FUNCTION_BLOCK FB_OmronLD90 EXTENDS FB_ROB_AMR IMPLEMENTS 
VAR_INPUT
END_VAR
VAR_OUTPUT
END_VAR
VAR
	//Reference to Skills

END_VAR

StateMachine(); // Method in FB_Base
ComMachine();	//Method in FB_ROB
DBClient();	//Datenbank Client in FB_ROB


PiNPl(Rob:=ADR(THIS^));

METHOD ComMachine : BOOL
VAR_INPUT
END_VAR
CASE eConnectionState OF


    // =========================================================
    // DISCONNECTED
    // =========================================================

    eCommunicationState.DISCONNECTED:

       _connected := FALSE;


        // Make sure socket handle is cleared
//         hSocket


        // -----------------------------------------------------
        // Connect requested
        // -----------------------------------------------------

        IF xConnectRequest THEN

            xConnectRequest := FALSE;

            // Clear previous errors
            Error := FALSE;
            ErrorId := 0;
            SocketErrorId := 0;

            // Start FB_SocketConnect
            xSocketConnectExecute := TRUE;

            eConnectionState :=
                eCommunicationState.CONNECTING;

        END_IF;


    // =========================================================
    // CONNECTING
    // =========================================================

    eCommunicationState.CONNECTING:

        _connected := FALSE;
        


        // -----------------------------------------------------
        // Execute FB_SocketConnect
        // -----------------------------------------------------

        fbSocketConnect(
            sSrvNetId := '',
            sRemoteHost := ComConfig.sIpAddress,
            nRemotePort := ComConfig.nPort,
            bExecute := xSocketConnectExecute,
            tTimeout := ComConfig.tTimeout
        );


        // Execute must only be TRUE for one cycle
        xSocketConnectExecute := FALSE;


        // -----------------------------------------------------
        // Connection successful
        // -----------------------------------------------------

        IF NOT fbSocketConnect.bBusy
            AND NOT fbSocketConnect.bError
//             AND (fbSocketConnect.hSocket <> 0)
        THEN

            hSocket :=
                fbSocketConnect.hSocket;

            _connected := TRUE;
    

            Error := FALSE;
            ErrorId := 0;
            SocketErrorId := 0;

            eConnectionState :=
                eCommunicationState.CONNECTED;

        END_IF;


        // -----------------------------------------------------
        // Connection failed
        // -----------------------------------------------------

        IF NOT fbSocketConnect.bBusy
            AND fbSocketConnect.bError
        THEN

            _connected := FALSE;

            Error := TRUE;

            SocketErrorId :=
                fbSocketConnect.nErrId;

            ErrorId :=
                fbSocketConnect.nErrId;

//             hSocket := 0;

            eConnectionState :=
                eCommunicationState.ERROR;

        END_IF;


    // =========================================================
    // CONNECTED
    // =========================================================

    eCommunicationState.CONNECTED:

        _connected := TRUE;



        // -----------------------------------------------------
        // Disconnect requested
        // -----------------------------------------------------

        IF xDisconnectRequest THEN

            xDisconnectRequest := FALSE;


            // Start socket close
            xSocketCloseExecute := TRUE;

            eConnectionState :=
                eCommunicationState.DISCONNECTING;

        END_IF;


    // =========================================================
    // DISCONNECTING
    // =========================================================

    eCommunicationState.DISCONNECTING:

        _connected := FALSE;


        // -----------------------------------------------------
        // Execute FB_SocketClose
        // -----------------------------------------------------

        fbSocketClose(
            sSrvNetId := '',
            hSocket := hSocket,
            bExecute := xSocketCloseExecute,
            tTimeout := ComConfig.tTimeout
        );


        // Execute only for one cycle
        xSocketCloseExecute := FALSE;


        // -----------------------------------------------------
        // Socket closed successfully
        // -----------------------------------------------------

        IF NOT fbSocketClose.bBusy
            AND NOT fbSocketClose.bError
        THEN

            _connected := FALSE;


//             hSocket := 0;

            eConnectionState :=
                eCommunicationState.DISCONNECTED;

        END_IF;


        // -----------------------------------------------------
        // Socket close failed
        // -----------------------------------------------------

        IF NOT fbSocketClose.bBusy
            AND fbSocketClose.bError
        THEN

            _connected := FALSE;


            Error := TRUE;

            SocketErrorId :=
                fbSocketClose.nErrId;

            ErrorId :=
                fbSocketClose.nErrId;

            // The socket should no longer be used
//             hSocket := 0;

            eConnectionState :=
                eCommunicationState.ERROR;

        END_IF;


    // =========================================================
    // ERROR
    // =========================================================

    eCommunicationState.ERROR:

        _connected := FALSE;
        // -----------------------------------------------------
        // Do not attempt to use the socket after an error
        // -----------------------------------------------------

//         hSocket := 0;


        // -----------------------------------------------------
        // A new connection request can recover from the error
        // -----------------------------------------------------

        IF xConnectRequest THEN

            xConnectRequest := FALSE;

            Error := FALSE;
            ErrorId := 0;
            SocketErrorId := 0;

            xSocketConnectExecute := TRUE;

            eConnectionState :=
                eCommunicationState.CONNECTING;

        END_IF;


END_CASE;
END_METHOD

{warning 'Add method implementation '}
METHOD Connect : BOOL

Connect := FALSE;

// Already connected
IF eConnectionState = eCommunicationState.CONNECTED THEN
    Connect := TRUE;
    RETURN;
END_IF;

// Already trying to connect
IF eConnectionState = eCommunicationState.CONNECTING THEN
    Connect := TRUE;
    RETURN;
END_IF;

// Don't accept a new connection while disconnecting
IF eConnectionState = eCommunicationState.DISCONNECTING THEN
    RETURN;
END_IF;

// Validate address
IF LEN(ComConfig.sIpAddress) = 0 THEN
    Error := TRUE;
//     ErrorId := 16#1001;
    RETURN;
END_IF;

// Validate port
IF ComConfig.nPort = 0 THEN
    Error := TRUE;
//     ErrorId := 16#1002;
    RETURN;
END_IF;

// Clear previous error
Error := FALSE;
ErrorId := 0;

// Request connection
xConnectRequest := TRUE;

Connect := TRUE;
END_METHOD

{warning 'Add property implementation'}
PROPERTY Connected : BOOL
GET
Connected:=_connected;
END_GET
END_PROPERTY

{warning 'Add method implementation '}
METHOD Disconnect : BOOL
END_METHOD

METHOD Dock : BOOL
END_METHOD

{warning 'Add method implementation '}
METHOD FINAL GoToGoal : BOOL
VAR_INPUT
	Goal: STRING;
END_VAR
END_METHOD

{warning 'Add method implementation '}
METHOD GoToPoint : BOOL

VAR_INPUT
	rX, rY, rTheta: REAL;
END_VAR
END_METHOD

METHOD MC_ChangeSpeedOverride : INT
VAR_INPUT
	factor	: REAL;
END_VAR
END_METHOD

METHOD MC_MoveAxesAbsolute : BOOL
VAR_INPUT
	target	: stTarget3D;
END_VAR
END_METHOD

METHOD MC_MoveAxesRelative : BOOL
VAR_INPUT
	axes	: ARRAY [1..6] OF FB_Axis;
	offsets	: ARRAY [1..6] OF REAL;
END_VAR
END_METHOD

METHOD MC_MoveLinearAbsolute : BOOL
VAR_INPUT
	target	: stTarget3D;
END_VAR
END_METHOD

METHOD MC_ReadAnalogInput : LREAL
VAR_INPUT
	input	: INT;
END_VAR
END_METHOD

METHOD MC_ReadDigitalInput : BOOL
VAR_INPUT
	input	: INT;
END_VAR
END_METHOD

METHOD MC_SetDigitalOutput : BOOL
VAR_INPUT
	output	: INT;
	value	: BOOL;
END_VAR
END_METHOD

METHOD MC_SetOperationMode : BOOL
VAR_INPUT
	mode	: eMode;
END_VAR
END_METHOD

METHOD onActivate : BOOL
// ---- Init ----
transitionresult:=eResult.None;



// ---- Change ----

// _mode:= eMode.Automatic;




// ---- Check ----
transitionresult := eResult.SUCCESS;

IF Error THEN
	transitionresult:= eResult.ERROR;
END_IF


// ---- Change State ----
IF transitionresult= eResult.SUCCESS THEN
	State:=eState.Active;
ELSIF transitionresult= eResult.FAILURE THEN
	State:=eState.Inactive;
ELSIF transitionresult= eResult.ERROR THEN
	State:=eState.ErrorProcessing;
ELSE
	ADSLOGSTR(ADSLOG_MSGTYPE_WARN,'Transitionresult from onActivate is None','');
END_IF
END_METHOD

METHOD onCleanup : BOOL
// ---- Init ----
transitionresult:=eResult.None;



// ---- Change ----

IF Connected THEN
	Disconnect();
END_IF





// ---- Check ----
transitionresult := eResult.SUCCESS;


// ---- Change State ----
IF transitionresult= eResult.SUCCESS THEN
	State:=eState.Unconfigured;
ELSIF transitionresult= eResult.FAILURE THEN
	ADSLOGSTR(ADSLOG_MSGTYPE_WARN,'Transitionresult from onCleanup is FAILURE ','');
ELSIF transitionresult= eResult.ERROR THEN
	State:=eState.ErrorProcessing;
ELSE
	ADSLOGSTR(ADSLOG_MSGTYPE_WARN,'Transitionresult from onCleanup is NONE','');
END_IF
END_METHOD

METHOD onConfigure : BOOL
// ---- Init ----
transitionresult:=eResult.None;



// ---- Change ----

Connect();




// ---- Check ----
IF Connected THEN
	transitionresult := eResult.SUCCESS;
ELSE
	transitionresult := eResult.FAILURE;
END_IF

IF Error THEN
	transitionresult:= eResult.ERROR;
END_IF



// ---- Change State ----
IF transitionresult= eResult.SUCCESS THEN
	State:=eState.Inactive;
ELSIF transitionresult= eResult.FAILURE THEN
	State:=eState.Unconfigured;
ELSIF transitionresult= eResult.ERROR THEN
	State:=eState.ErrorProcessing;
ELSE
	ADSLOGSTR(ADSLOG_MSGTYPE_WARN,'Transitionresult from onConfigure is None','');
END_IF
END_METHOD

METHOD onDeactivate : BOOL
// ---- Init ----
transitionresult:=eResult.None;



// ---- Change ----

// _mode:= eMode.Manual;




// ---- Check ----
transitionresult := eResult.SUCCESS;

IF Error THEN
	transitionresult:= eResult.ERROR;
END_IF

// ---- Change State ----
IF transitionresult= eResult.SUCCESS THEN
	State:=eState.Inactive;
ELSIF transitionresult= eResult.FAILURE THEN
	ADSLOGSTR(ADSLOG_MSGTYPE_WARN,'Transitionresult from onDeactivate is FAILURE','');
ELSIF transitionresult= eResult.ERROR THEN
	State:=eState.ErrorProcessing;
ELSE
	ADSLOGSTR(ADSLOG_MSGTYPE_WARN,'Transitionresult from onDeactivate is None','');
END_IF
END_METHOD

METHOD onError : BOOL
// ---- Init ----
transitionresult:=eResult.None;



// ---- Change ----

// _mode:= eMode.Manual;




// ---- Check ----
transitionresult := eResult.SUCCESS;


// ---- Change State ----
IF transitionresult= eResult.SUCCESS THEN
	State:=eState.Unconfigured;
ELSIF transitionresult= eResult.FAILURE THEN
	State:=eState.Finalized;
ELSIF transitionresult= eResult.ERROR THEN
	ADSLOGSTR(ADSLOG_MSGTYPE_WARN,'Transitionresult from onError is Error','');
ELSE
	ADSLOGSTR(ADSLOG_MSGTYPE_WARN,'Transitionresult from onError is None','');
END_IF
END_METHOD

METHOD onShutdown : BOOL
// ---- Init ----
transitionresult:=eResult.None;



// ---- Change ----

// _mode:= eMode.Manual;

IF Connected THEN
	Disconnect();
END_IF


// ---- Check ----
transitionresult := eResult.SUCCESS;

IF Error THEN
	transitionresult:= eResult.ERROR;
END_IF

// ---- Change State ----
IF transitionresult= eResult.SUCCESS THEN
	State:=eState.Finalized;
ELSIF transitionresult= eResult.FAILURE THEN
	ADSLOGSTR(ADSLOG_MSGTYPE_WARN,'Transitionresult from onShutdown is FAILURE','');
ELSIF transitionresult= eResult.ERROR THEN
	State:=eState.ErrorProcessing;
ELSE
	ADSLOGSTR(ADSLOG_MSGTYPE_WARN,'Transitionresult from onShutdown is None','');
END_IF
END_METHOD

{warning 'Add method implementation '}
METHOD ResetConnection : BOOL
END_METHOD

{warning 'Add method implementation '}
METHOD Undock : BOOL
END_METHOD

END_FUNCTION_BLOCK

(* stored: Version 1.1.0.1, ProductVersion 3.1.4026.18
   POU FB_OmronLD90: Id {fac74160-c2b3-4f77-bd69-eddf1970c653}, SpecialFunc None
   Folder Communication: Id {2a9c337e-719c-4121-a5a9-4ddfd8584a43}
   Folder MotionControl: Id {94b27a46-e651-4eff-a38f-a2a3d5ee10b5}
   Folder StateControl: Id {67994def-610e-4a0b-a6c8-85df31e22884}
   Method ComMachine: Id {040d86b8-c78e-42d4-a5c1-25c0270b6e14}
   Method Connect: Id {70fa978a-67c6-43be-99fb-d03c8689cf07}
   Property Connected: Id {e71d8962-d52b-46f4-b79d-88e001b39f65}
   Get Get: Id {1724321d-02c7-40cd-942a-414eba41ba06}
   Method Disconnect: Id {c75c2374-9ebb-4dd8-a5bc-f61f0a69c931}
   Method Dock: Id {ed889dfa-89d4-4c82-aa20-11f1706e94ee}
   Method GoToGoal: Id {bbbc983d-cf30-4dcf-8a44-55f25ea52986}
   Method GoToPoint: Id {dc0441f1-6bc0-484a-9b38-d363d0c2594e}
   Method MC_ChangeSpeedOverride: Id {713f1143-5191-40a4-b72a-885f3f7f8583}
   Method MC_MoveAxesAbsolute: Id {0cd522ad-3196-4d60-88fa-579c31568d4a}
   Method MC_MoveAxesRelative: Id {f73d189b-ff87-4fed-aa85-efb29eda32d4}
   Method MC_MoveLinearAbsolute: Id {ca83c178-9848-4cc0-b00b-256b7c7dfbf1}
   Method MC_ReadAnalogInput: Id {f0ca8b75-c40b-4e48-971c-e8720e2a2c9d}
   Method MC_ReadDigitalInput: Id {c7317b25-d839-47d8-b4be-44cfbee742a7}
   Method MC_SetDigitalOutput: Id {91ad8e1f-9be7-4585-b174-cb9248903477}
   Method MC_SetOperationMode: Id {41d82623-631b-48fe-bc0b-275e5972c6a7}
   Method onActivate: Id {7fa92802-2ede-4193-9973-ad7754d17239}
   Method onCleanup: Id {7747948a-f8e1-4cdb-8a20-610ab536a0ef}
   Method onConfigure: Id {c568c508-6321-435c-b7c4-683ad73a8f42}
   Method onDeactivate: Id {57ce1156-6b80-40b7-8fff-100660e6e779}
   Method onError: Id {74c0a508-94ea-4785-a0ea-1af2639ff5e5}
   Method onShutdown: Id {f496723a-9c1c-413c-b4ed-4d78c56c0863}
   Method ResetConnection: Id {1a6fc39d-923f-4cb8-bc55-cd413f8ec29d}
   Method Undock: Id {ad3375f8-7552-4141-bde9-a85c6d9963c4} *)
